% RSLogix 500 project G01098.RSS, saved by version 8.10.00.18 %
PROJECT "G01098"    % processor: SLC 500, 1747-L542 %

PROGRAM FILES
  LAD 2   30 rungs
  LAD 4   21 rungs
  LAD 5   16 rungs
  LAD 20   18 rungs
  LAD 25   24 rungs
  LAD 28   18 rungs
  LAD 29   60 rungs
  LAD 30   13 rungs
  LAD 31   63 rungs
  LAD 32   32 rungs
  LAD 33   10 rungs
  LAD 34   57 rungs
  LAD 35   6 rungs
  LAD 36   5 rungs
  LAD 37   16 rungs
  LAD 38   18 rungs
  LAD 39   59 rungs
  LAD 40   66 rungs
  LAD 50   21 rungs
  LAD 75   16 rungs
  LAD 77   16 rungs
  LAD 80   16 rungs
  LAD 85   37 rungs
  LAD 100   11 rungs
  LAD 101   13 rungs
  LAD 102   14 rungs
  LAD 103   3 rungs
  LAD 110   5 rungs
  LAD 200   24 rungs

DATA FILES
  O0 OUTPUT  23 elements
  I1 INPUT  19 elements
  S2 STATUS  164 elements
  B3 BINARY  105 elements
  T4 TIMER  91 elements
  C5 COUNTER  10 elements
  R6 CONTROL  1 elements
  N7 INTEGER  110 elements
  F8 FLOAT  10 elements
  N10   100 elements
  N11   100 elements
  F15   20 elements
  N20   30 elements
  N30   70 elements
  B33   5 elements
  B34   5 elements
  B50   100 elements
  B51   50 elements
  N52   70 elements
  N53   100 elements
  F54   10 elements
  F55   10 elements
  B56   1 elements
  N58   20 elements
  N59   134 elements
  N60   15 elements
  N61   30 elements
  B94   1 elements
  B95   1 elements
  B96   1 elements
  B97   1 elements
  B98   1 elements
  B99   1 elements
  F197   22 elements
  F198   22 elements
  F199   22 elements
  F200   22 elements
  F201   22 elements
  F202   22 elements
  F203   22 elements
  F204   22 elements
  F205   22 elements
  F206   22 elements
  F207   22 elements
  F208   22 elements
  F209   22 elements
  F210   22 elements
  F211   22 elements
  F212   22 elements
  F213   22 elements
  F214   22 elements
  F215   22 elements
  F216   22 elements
  F217   22 elements
  F218   22 elements
  F219   22 elements
  F220   22 elements
  F221   22 elements
  F222   22 elements
  F223   22 elements
  F224   22 elements
  F225   22 elements
  F226   22 elements
  F227   22 elements
  F228   22 elements
  F229   22 elements
  F230   22 elements
  F231   22 elements
  F232   22 elements
  F233   22 elements
  F234   22 elements
  F235   22 elements
  F236   22 elements
  F237   22 elements
  F238   22 elements
  F239   22 elements
  F240   22 elements
  F241   22 elements
  F242   22 elements
  F243   22 elements
  F244   22 elements
  F245   22 elements
  F246   22 elements
  F247   22 elements
  F248   22 elements
  F249   22 elements
  F250   22 elements

LADDER 2
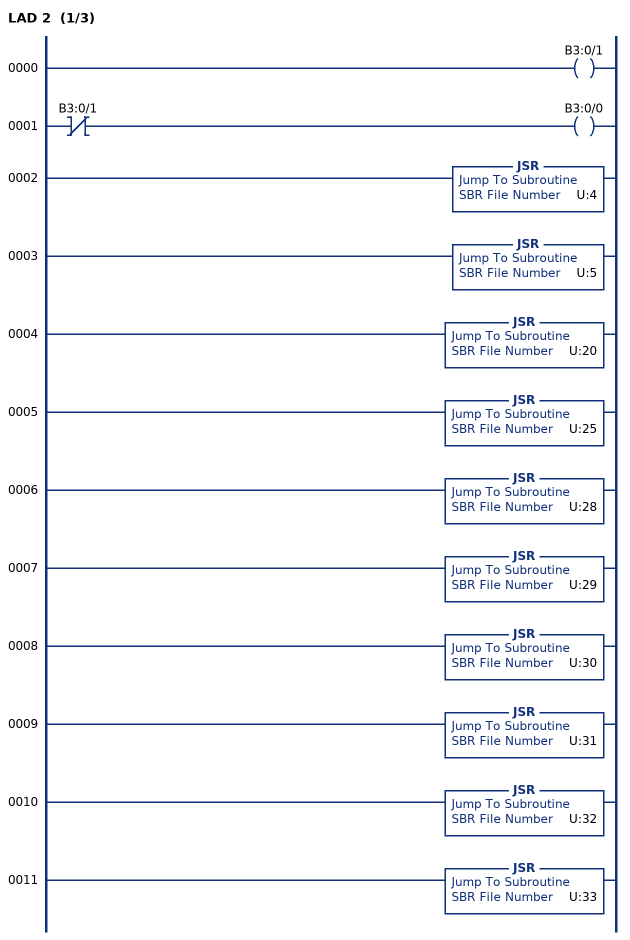
% Rung: 0 %
SOR OTE B3:0/1 EOR
% Rung: 1 %
SOR XIO B3:0/1 OTE B3:0/0 EOR
% Rung: 2 %
SOR JSR U:4 EOR
% Rung: 3 %
SOR JSR U:5 EOR
% Rung: 4 %
SOR JSR U:20 EOR
% Rung: 5 %
SOR JSR U:25 EOR
% Rung: 6 %
SOR JSR U:28 EOR
% Rung: 7 %
SOR JSR U:29 EOR
% Rung: 8 %
SOR JSR U:30 EOR
% Rung: 9 %
SOR JSR U:31 EOR
% Rung: 10 %
SOR JSR U:32 EOR
% Rung: 11 %
SOR JSR U:33 EOR

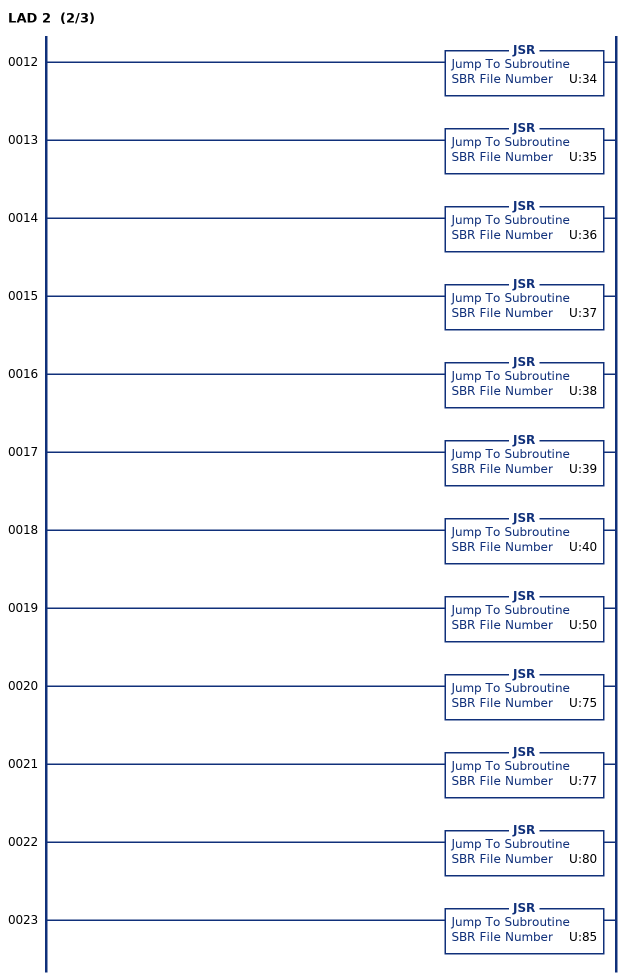
% Rung: 12 %
SOR JSR U:34 EOR
% Rung: 13 %
SOR JSR U:35 EOR
% Rung: 14 %
SOR JSR U:36 EOR
% Rung: 15 %
SOR JSR U:37 EOR
% Rung: 16 %
SOR JSR U:38 EOR
% Rung: 17 %
SOR JSR U:39 EOR
% Rung: 18 %
SOR JSR U:40 EOR
% Rung: 19 %
SOR JSR U:50 EOR
% Rung: 20 %
SOR JSR U:75 EOR
% Rung: 21 %
SOR JSR U:77 EOR
% Rung: 22 %
SOR JSR U:80 EOR
% Rung: 23 %
SOR JSR U:85 EOR

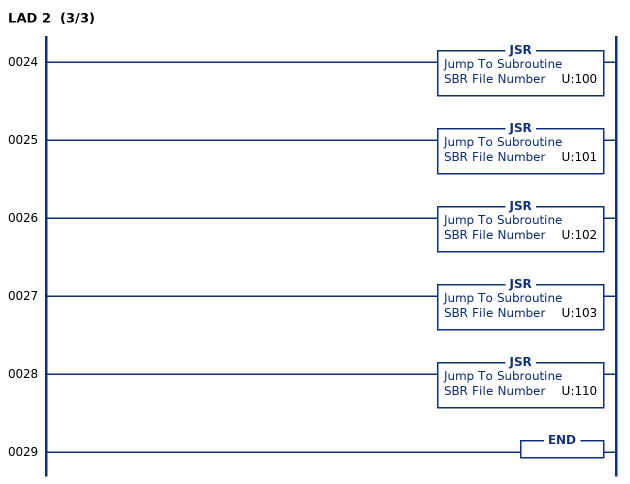
% Rung: 24 %
SOR JSR U:100 EOR
% Rung: 25 %
SOR JSR U:101 EOR
% Rung: 26 %
SOR JSR U:102 EOR
% Rung: 27 %
SOR JSR U:103 EOR
% Rung: 28 %
SOR JSR U:110 EOR
% Rung: 29 %
SOR END EOR

LADDER 4
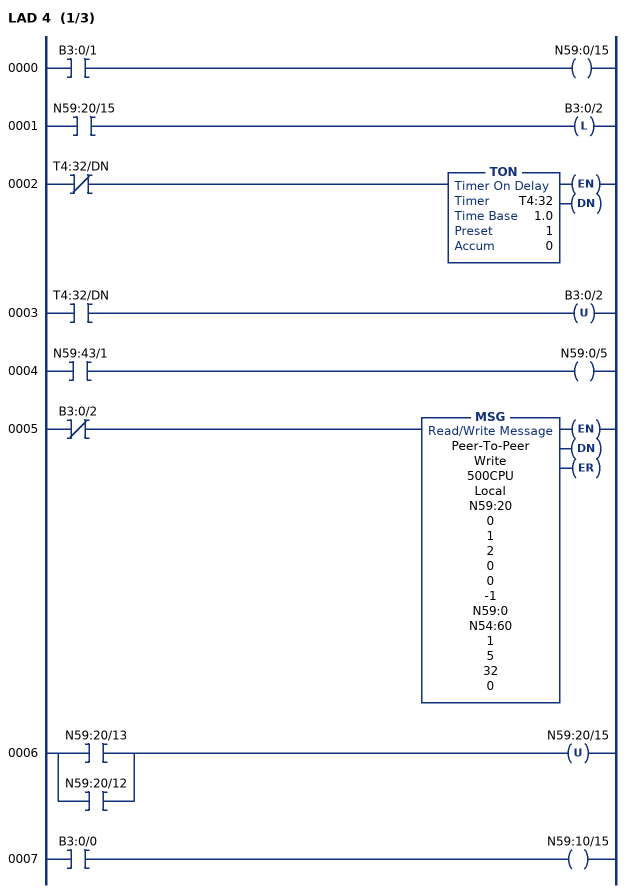
% Rung: 0 %
SOR XIC B3:0/1 OTE N59:0/15 EOR
% Rung: 1 %
SOR XIC N59:20/15 OTL B3:0/2 EOR
% Rung: 2 %
SOR XIO T4:32/DN TON T4:32 1.0 1 0 EOR
% Rung: 3 %
SOR XIC T4:32/DN OTU B3:0/2 EOR
% Rung: 4 %
SOR XIC N59:43/1 OTE N59:0/5 EOR
% Rung: 5 %
SOR XIO B3:0/2 MSG Peer-To-Peer Write 500CPU Local N59:20 0 1 2 0 0 -1 N59:0 N54:60 1 5 32 0 EOR
%   MSG set-up: 500CPU Write | 5 | 1 | N54:60 | N59:0 | 0 | 2 | 2 | CLIENT | 0 | 0 %
% Rung: 6 %
SOR BST XIC N59:20/13 NXB XIC N59:20/12 BND OTU N59:20/15 EOR
% Rung: 7 %
SOR XIC B3:0/0 OTE N59:10/15 EOR

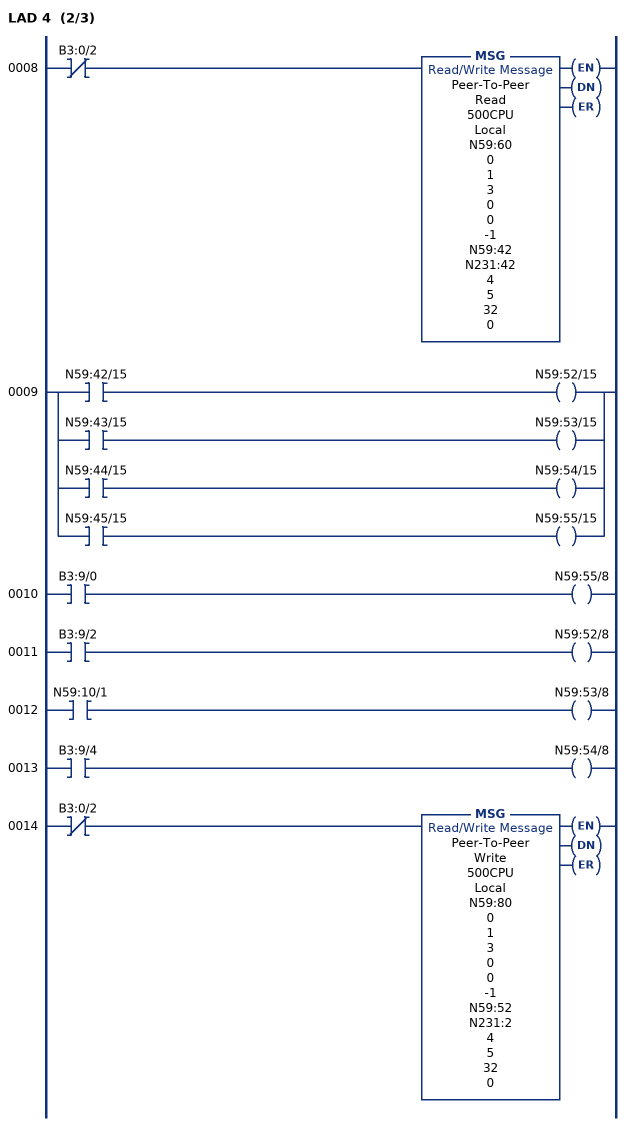
% Rung: 8 %
SOR XIO B3:0/2 MSG Peer-To-Peer Read 500CPU Local N59:60 0 1 3 0 0 -1 N59:42 N231:42 4 5 32 0 EOR
%   MSG set-up: 500CPU Read | 5 | 4 | N231:42 | N59:42 | 0 | 3 | 3 | CLIENT | 0 | 0 %
% Rung: 9 %
SOR BST XIC N59:42/15 OTE N59:52/15 NXB XIC N59:43/15 OTE N59:53/15 NXB XIC N59:44/15 OTE N59:54/15 NXB XIC N59:45/15 OTE N59:55/15 BND EOR
% Rung: 10 %
SOR XIC B3:9/0 OTE N59:55/8 EOR
% Rung: 11 %
SOR XIC B3:9/2 OTE N59:52/8 EOR
% Rung: 12 %
SOR XIC N59:10/1 OTE N59:53/8 EOR
% Rung: 13 %
SOR XIC B3:9/4 OTE N59:54/8 EOR
% Rung: 14 %
SOR XIO B3:0/2 MSG Peer-To-Peer Write 500CPU Local N59:80 0 1 3 0 0 -1 N59:52 N231:2 4 5 32 0 EOR
%   MSG set-up: 500CPU Write | 5 | 4 | N231:2 | N59:52 | 0 | 3 | 3 | CLIENT | 0 | 0 %

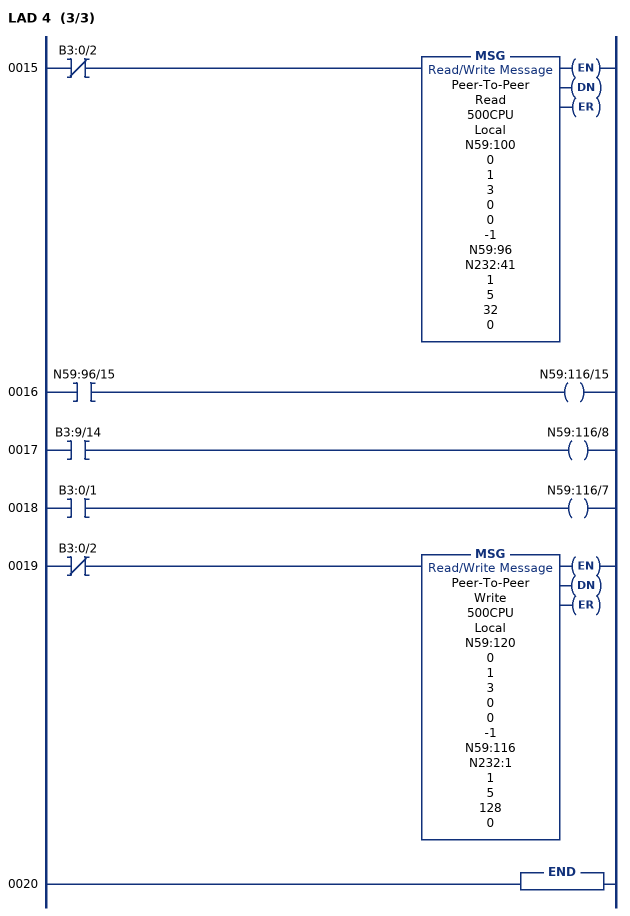
% Rung: 15 %
SOR XIO B3:0/2 MSG Peer-To-Peer Read 500CPU Local N59:100 0 1 3 0 0 -1 N59:96 N232:41 1 5 32 0 EOR
%   MSG set-up: 500CPU Read | 5 | 1 | N232:41 | N59:96 | 0 | 3 | 3 | CLIENT | 0 | 0 %
% Rung: 16 %
SOR XIC N59:96/15 OTE N59:116/15 EOR
% Rung: 17 %
SOR XIC B3:9/14 OTE N59:116/8 EOR
% Rung: 18 %
SOR XIC B3:0/1 OTE N59:116/7 EOR
% Rung: 19 %
SOR XIO B3:0/2 MSG Peer-To-Peer Write 500CPU Local N59:120 0 1 3 0 0 -1 N59:116 N232:1 1 5 128 0 EOR
%   MSG set-up: 500CPU Write | 5 | 1 | N232:1 | N59:116 | 0 | 3 | 3 | CLIENT | 0 | 0 %
% Rung: 20 %
SOR END EOR

LADDER 5
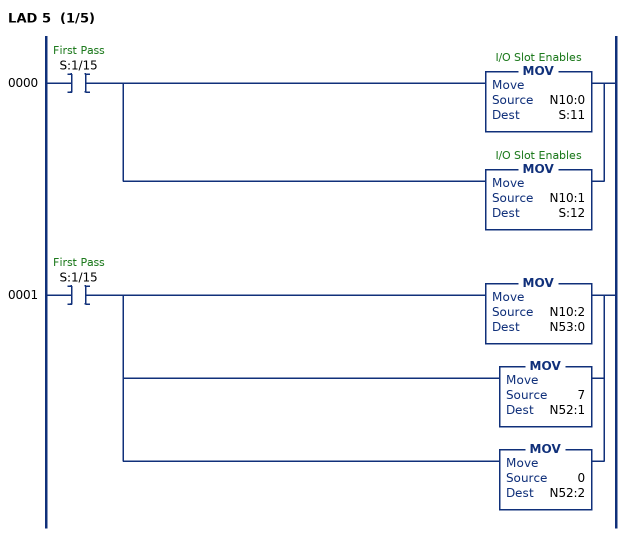
% Rung: 0 %
SOR XIC S:1/15 BST MOV N10:0 S:11 NXB MOV N10:1 S:12 BND EOR
%   S:1/15  "First Pass" %
%   S:11  "I/O Slot Enables" %
%   S:12  "I/O Slot Enables" %
% Rung: 1 %
SOR XIC S:1/15 BST MOV N10:2 N53:0 NXB MOV 7 N52:1 NXB MOV 0 N52:2 BND EOR
%   S:1/15  "First Pass" %

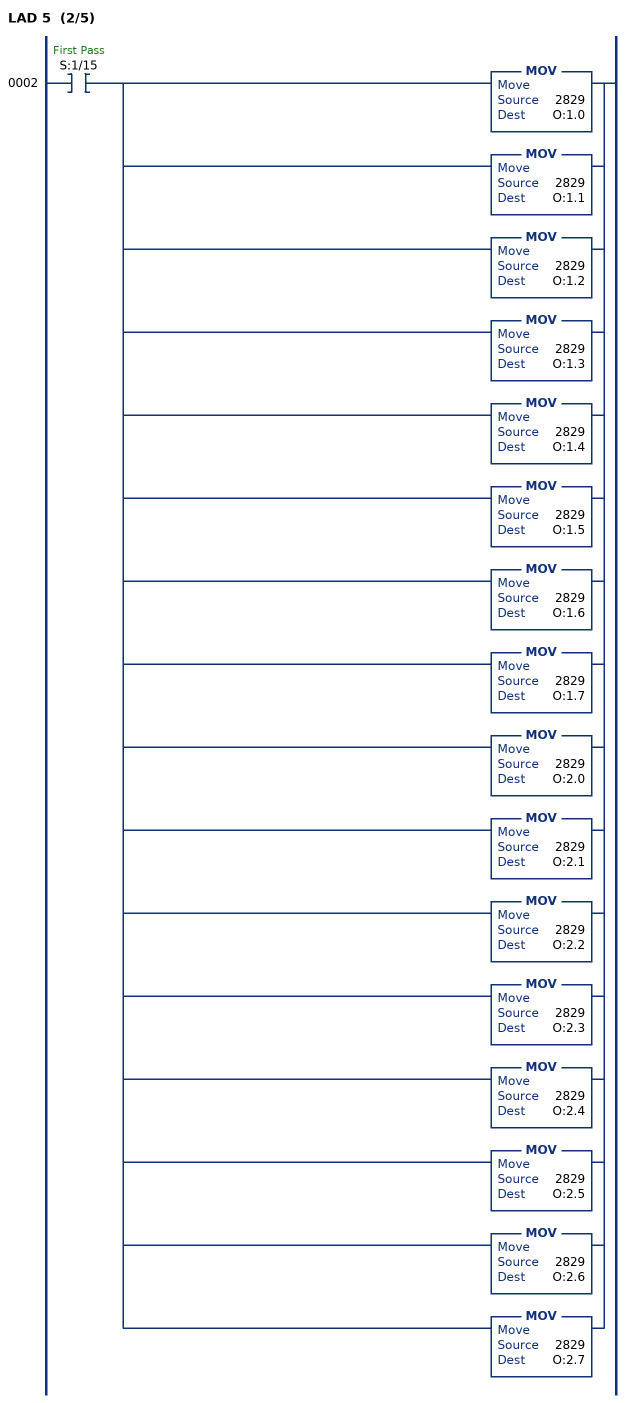
% Rung: 2 %
SOR XIC S:1/15 BST MOV 2829 O:1.0 NXB MOV 2829 O:1.1 NXB MOV 2829 O:1.2 NXB MOV 2829 O:1.3 NXB MOV 2829 O:1.4 NXB MOV 2829 O:1.5 NXB MOV 2829 O:1.6 NXB MOV 2829 O:1.7 NXB MOV 2829 O:2.0 NXB MOV 2829 O:2.1 NXB MOV 2829 O:2.2 NXB MOV 2829 O:2.3 NXB MOV 2829 O:2.4 NXB MOV 2829 O:2.5 NXB MOV 2829 O:2.6 NXB MOV 2829 O:2.7 BND EOR
%   S:1/15  "First Pass" %

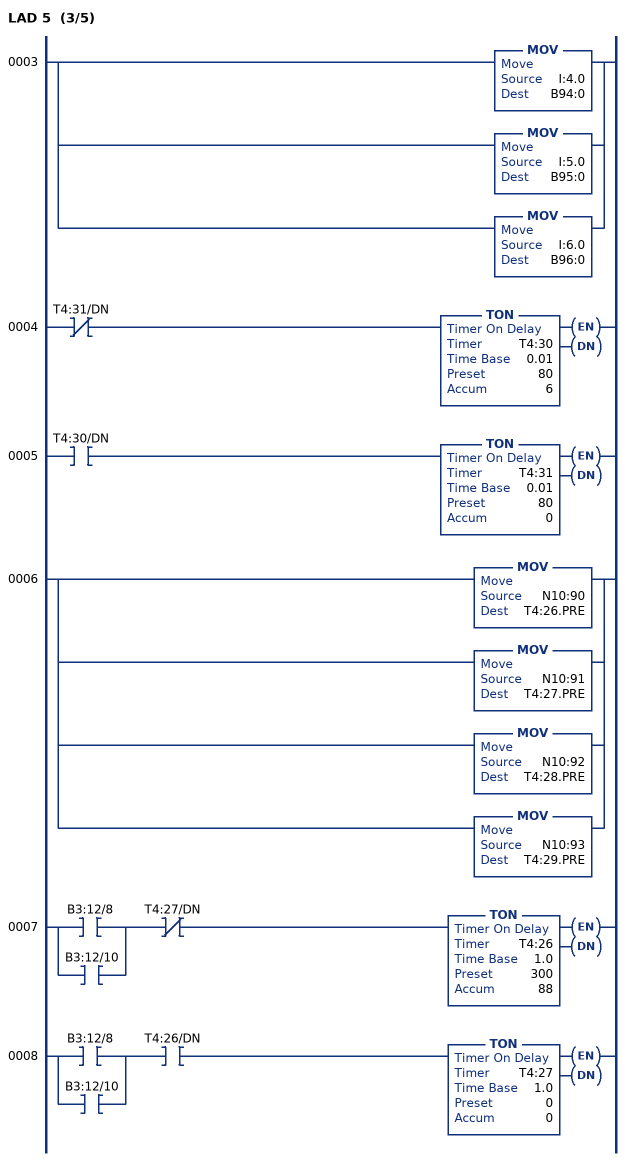
% Rung: 3 %
SOR BST MOV I:4.0 B94:0 NXB MOV I:5.0 B95:0 NXB MOV I:6.0 B96:0 BND EOR
% Rung: 4 %
SOR XIO T4:31/DN TON T4:30 0.01 80 6 EOR
% Rung: 5 %
SOR XIC T4:30/DN TON T4:31 0.01 80 0 EOR
% Rung: 6 %
SOR BST MOV N10:90 T4:26.PRE NXB MOV N10:91 T4:27.PRE NXB MOV N10:92 T4:28.PRE NXB MOV N10:93 T4:29.PRE BND EOR
% Rung: 7 %
SOR BST XIC B3:12/8 NXB XIC B3:12/10 BND XIO T4:27/DN TON T4:26 1.0 300 88 EOR
% Rung: 8 %
SOR BST XIC B3:12/8 NXB XIC B3:12/10 BND XIC T4:26/DN TON T4:27 1.0 0 0 EOR

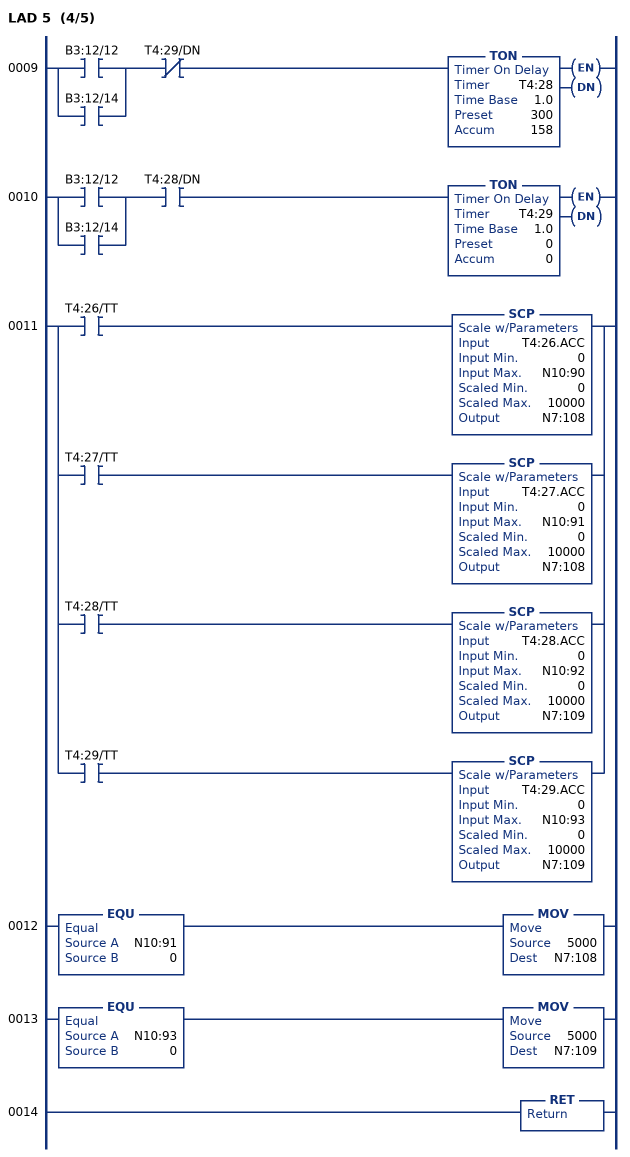
% Rung: 9 %
SOR BST XIC B3:12/12 NXB XIC B3:12/14 BND XIO T4:29/DN TON T4:28 1.0 300 158 EOR
% Rung: 10 %
SOR BST XIC B3:12/12 NXB XIC B3:12/14 BND XIC T4:28/DN TON T4:29 1.0 0 0 EOR
% Rung: 11 %
SOR BST XIC T4:26/TT SCP T4:26.ACC 0 N10:90 0 10000 N7:108 NXB XIC T4:27/TT SCP T4:27.ACC 0 N10:91 0 10000 N7:108 NXB XIC T4:28/TT SCP T4:28.ACC 0 N10:92 0 10000 N7:109 NXB XIC T4:29/TT SCP T4:29.ACC 0 N10:93 0 10000 N7:109 BND EOR
% Rung: 12 %
SOR EQU N10:91 0 MOV 5000 N7:108 EOR
% Rung: 13 %
SOR EQU N10:93 0 MOV 5000 N7:109 EOR
% Rung: 14 %
SOR RET EOR

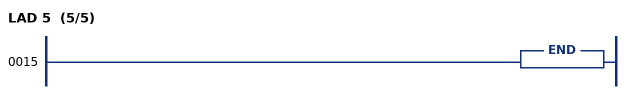
% Rung: 15 %
SOR END EOR

LADDER 20
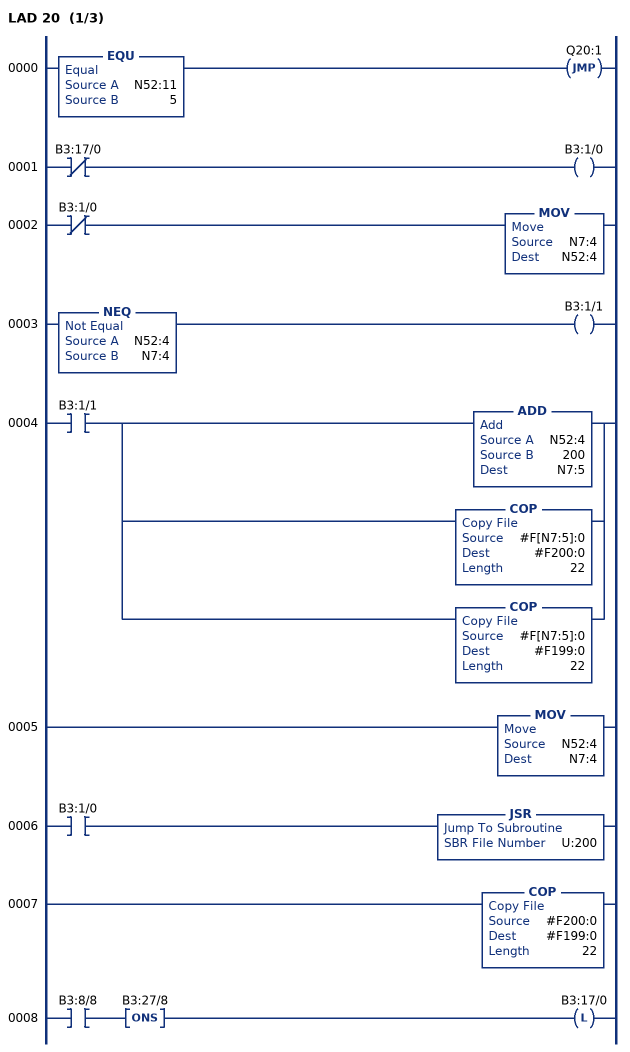
% Rung: 0 %
SOR EQU N52:11 5 JMP Q20:1 EOR
% Rung: 1 %
SOR XIO B3:17/0 OTE B3:1/0 EOR
% Rung: 2 %
SOR XIO B3:1/0 MOV N7:4 N52:4 EOR
% Rung: 3 %
SOR NEQ N52:4 N7:4 OTE B3:1/1 EOR
% Rung: 4 %
SOR XIC B3:1/1 BST ADD N52:4 200 N7:5 NXB COP #F[N7:5]:0 #F200:0 22 NXB COP #F[N7:5]:0 #F199:0 22 BND EOR
% Rung: 5 %
SOR MOV N52:4 N7:4 EOR
% Rung: 6 %
SOR XIC B3:1/0 JSR U:200 EOR
% Rung: 7 %
SOR COP #F200:0 #F199:0 22 EOR
% Rung: 8 %
SOR XIC B3:8/8 OSR B3:27/8 OTL B3:17/0 EOR

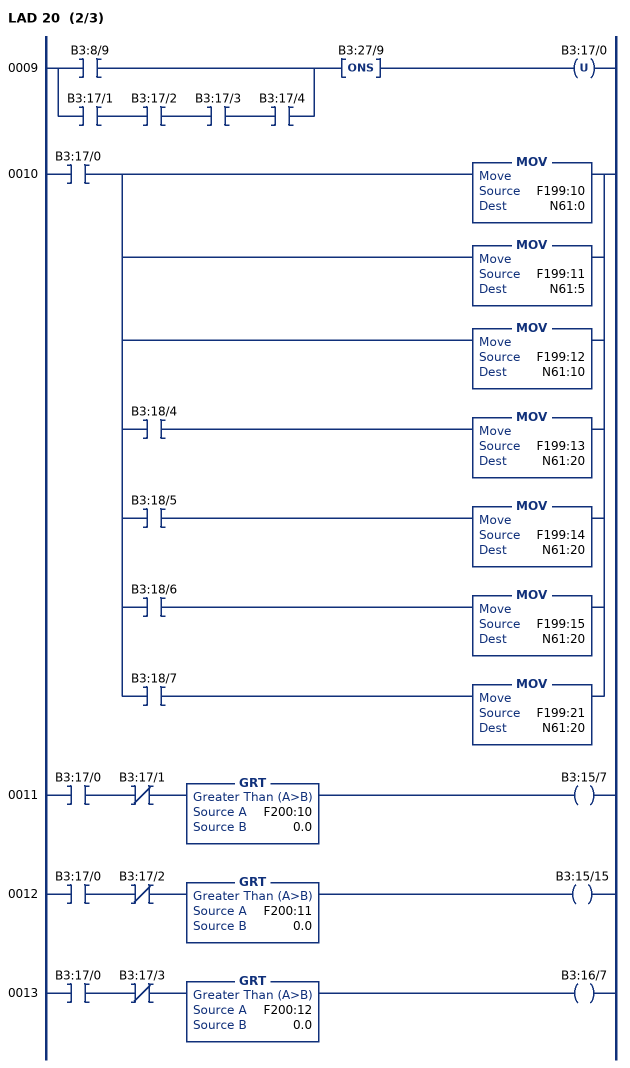
% Rung: 9 %
SOR BST XIC B3:8/9 NXB XIC B3:17/1 XIC B3:17/2 XIC B3:17/3 XIC B3:17/4 BND OSR B3:27/9 OTU B3:17/0 EOR
% Rung: 10 %
SOR XIC B3:17/0 BST MOV F199:10 N61:0 NXB MOV F199:11 N61:5 NXB MOV F199:12 N61:10 NXB XIC B3:18/4 MOV F199:13 N61:20 NXB XIC B3:18/5 MOV F199:14 N61:20 NXB XIC B3:18/6 MOV F199:15 N61:20 NXB XIC B3:18/7 MOV F199:21 N61:20 BND EOR
% Rung: 11 %
SOR XIC B3:17/0 XIO B3:17/1 GRT F200:10 0.0 OTE B3:15/7 EOR
% Rung: 12 %
SOR XIC B3:17/0 XIO B3:17/2 GRT F200:11 0.0 OTE B3:15/15 EOR
% Rung: 13 %
SOR XIC B3:17/0 XIO B3:17/3 GRT F200:12 0.0 OTE B3:16/7 EOR

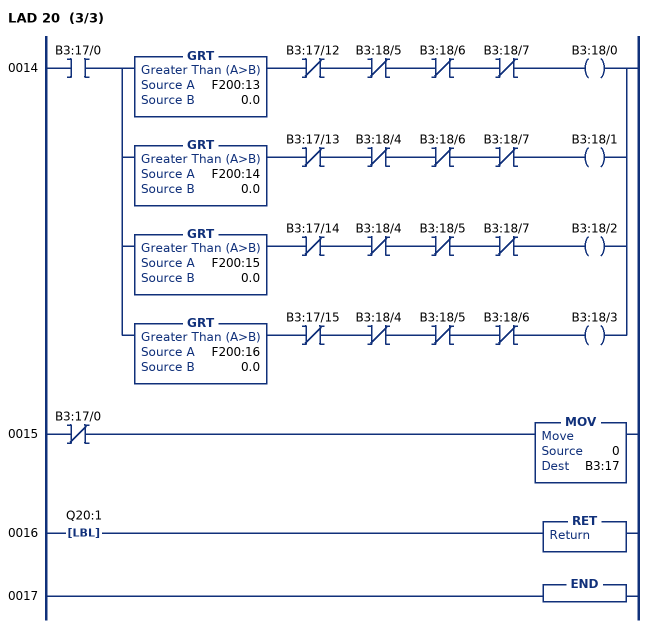
% Rung: 14 %
SOR XIC B3:17/0 BST GRT F200:13 0.0 XIO B3:17/12 XIO B3:18/5 XIO B3:18/6 XIO B3:18/7 OTE B3:18/0 NXB GRT F200:14 0.0 XIO B3:17/13 XIO B3:18/4 XIO B3:18/6 XIO B3:18/7 OTE B3:18/1 NXB GRT F200:15 0.0 XIO B3:17/14 XIO B3:18/4 XIO B3:18/5 XIO B3:18/7 OTE B3:18/2 NXB GRT F200:16 0.0 XIO B3:17/15 XIO B3:18/4 XIO B3:18/5 XIO B3:18/6 OTE B3:18/3 BND EOR
% Rung: 15 %
SOR XIO B3:17/0 MOV 0 B3:17 EOR
% Rung: 16 %
SOR LBL Q20:1 RET EOR
% Rung: 17 %
SOR END EOR

LADDER 25
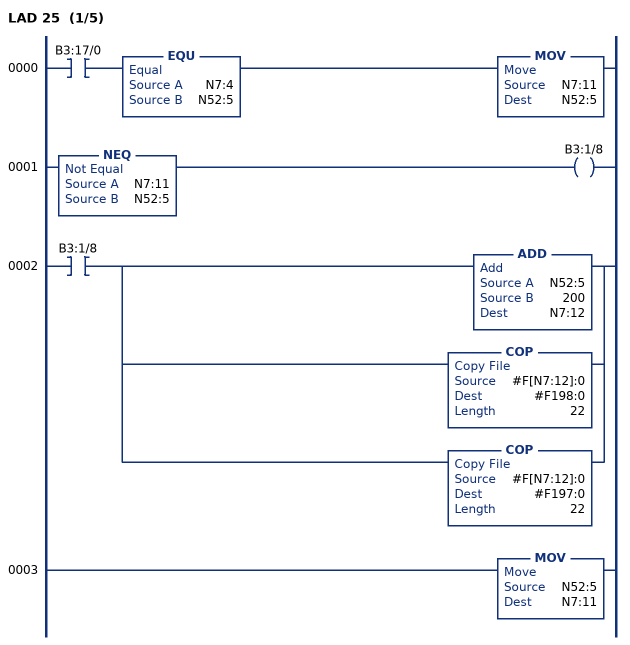
% Rung: 0 %
SOR XIC B3:17/0 EQU N7:4 N52:5 MOV N7:11 N52:5 EOR
% Rung: 1 %
SOR NEQ N7:11 N52:5 OTE B3:1/8 EOR
% Rung: 2 %
SOR XIC B3:1/8 BST ADD N52:5 200 N7:12 NXB COP #F[N7:12]:0 #F198:0 22 NXB COP #F[N7:12]:0 #F197:0 22 BND EOR
% Rung: 3 %
SOR MOV N52:5 N7:11 EOR

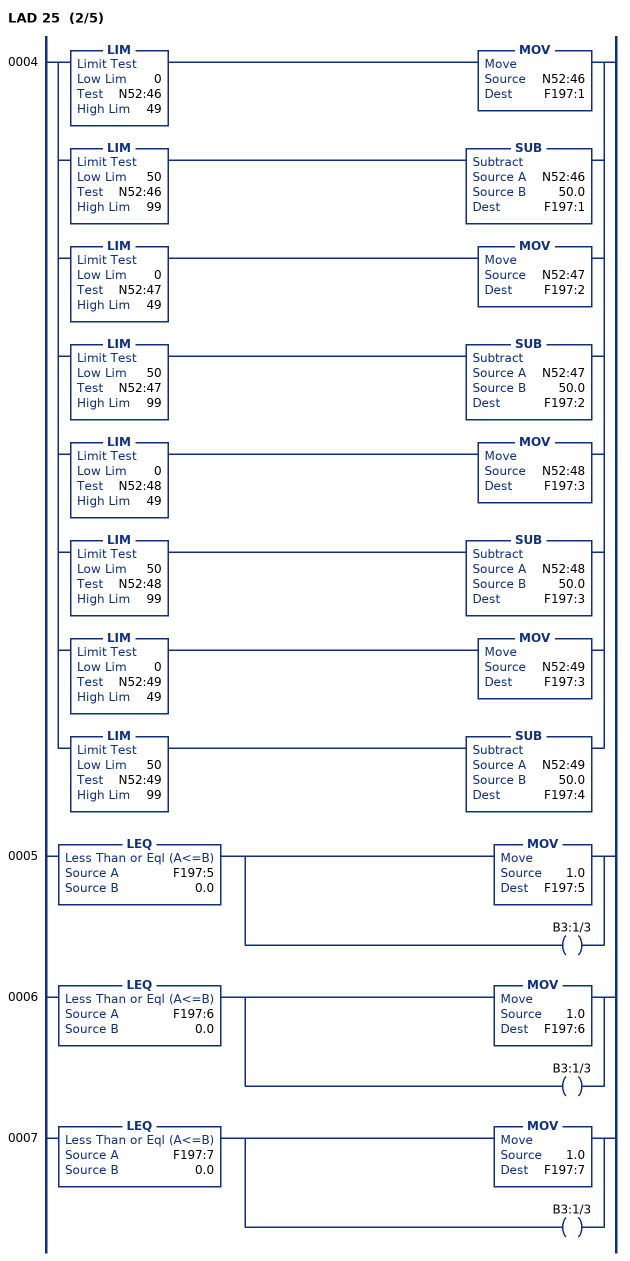
% Rung: 4 %
SOR BST LIM 0 N52:46 49 MOV N52:46 F197:1 NXB LIM 50 N52:46 99 SUB N52:46 50.0 F197:1 NXB LIM 0 N52:47 49 MOV N52:47 F197:2 NXB LIM 50 N52:47 99 SUB N52:47 50.0 F197:2 NXB LIM 0 N52:48 49 MOV N52:48 F197:3 NXB LIM 50 N52:48 99 SUB N52:48 50.0 F197:3 NXB LIM 0 N52:49 49 MOV N52:49 F197:3 NXB LIM 50 N52:49 99 SUB N52:49 50.0 F197:4 BND EOR
% Rung: 5 %
SOR LEQ F197:5 0.0 BST MOV 1.0 F197:5 NXB OTE B3:1/3 BND EOR
% Rung: 6 %
SOR LEQ F197:6 0.0 BST MOV 1.0 F197:6 NXB OTE B3:1/3 BND EOR
% Rung: 7 %
SOR LEQ F197:7 0.0 BST MOV 1.0 F197:7 NXB OTE B3:1/3 BND EOR

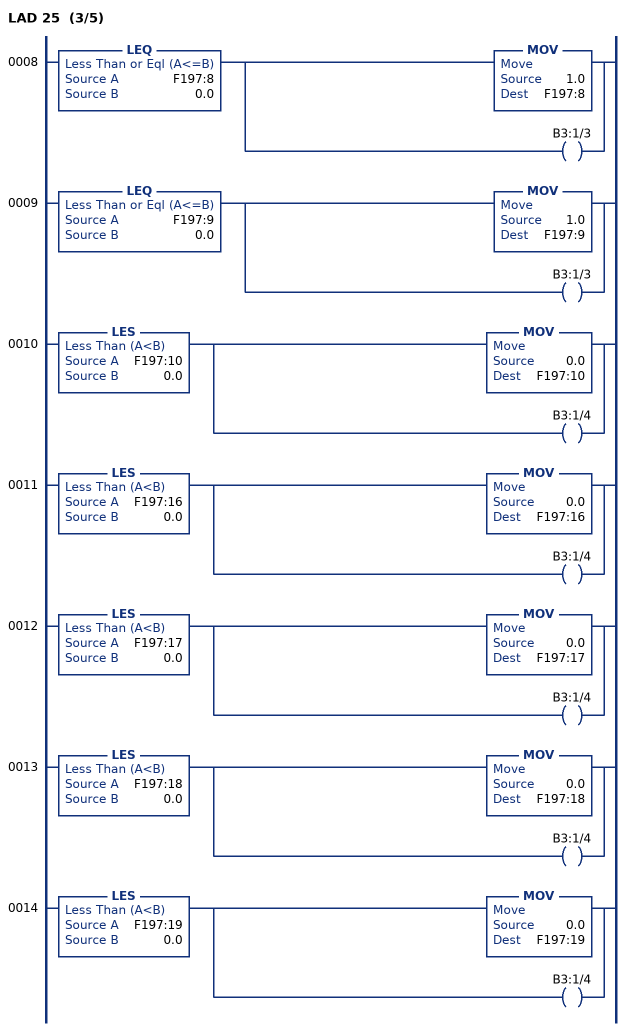
% Rung: 8 %
SOR LEQ F197:8 0.0 BST MOV 1.0 F197:8 NXB OTE B3:1/3 BND EOR
% Rung: 9 %
SOR LEQ F197:9 0.0 BST MOV 1.0 F197:9 NXB OTE B3:1/3 BND EOR
% Rung: 10 %
SOR LES F197:10 0.0 BST MOV 0.0 F197:10 NXB OTE B3:1/4 BND EOR
% Rung: 11 %
SOR LES F197:16 0.0 BST MOV 0.0 F197:16 NXB OTE B3:1/4 BND EOR
% Rung: 12 %
SOR LES F197:17 0.0 BST MOV 0.0 F197:17 NXB OTE B3:1/4 BND EOR
% Rung: 13 %
SOR LES F197:18 0.0 BST MOV 0.0 F197:18 NXB OTE B3:1/4 BND EOR
% Rung: 14 %
SOR LES F197:19 0.0 BST MOV 0.0 F197:19 NXB OTE B3:1/4 BND EOR

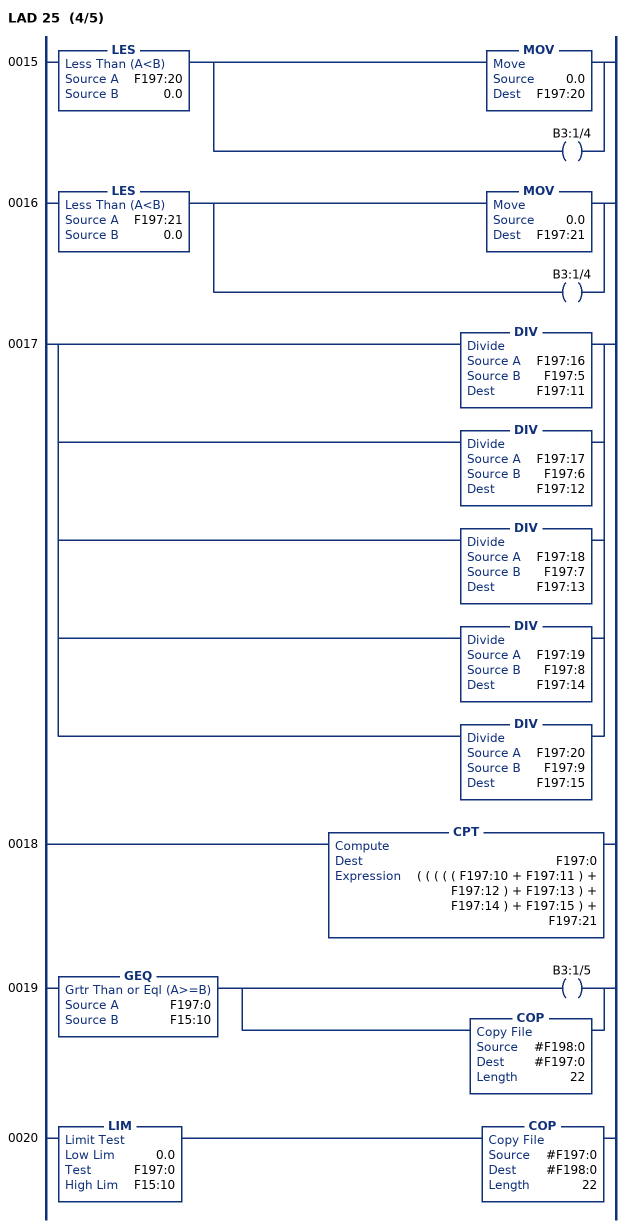
% Rung: 15 %
SOR LES F197:20 0.0 BST MOV 0.0 F197:20 NXB OTE B3:1/4 BND EOR
% Rung: 16 %
SOR LES F197:21 0.0 BST MOV 0.0 F197:21 NXB OTE B3:1/4 BND EOR
% Rung: 17 %
SOR BST DIV F197:16 F197:5 F197:11 NXB DIV F197:17 F197:6 F197:12 NXB DIV F197:18 F197:7 F197:13 NXB DIV F197:19 F197:8 F197:14 NXB DIV F197:20 F197:9 F197:15 BND EOR
% Rung: 18 %
SOR CPT F197:0 " ( ( ( ( ( F197:10 + F197:11 ) + F197:12 ) + F197:13 ) + F197:14 ) + F197:15 ) + F197:21 " EOR
% Rung: 19 %
SOR GEQ F197:0 F15:10 BST OTE B3:1/5 NXB COP #F198:0 #F197:0 22 BND EOR
% Rung: 20 %
SOR LIM 0.0 F197:0 F15:10 COP #F197:0 #F198:0 22 EOR

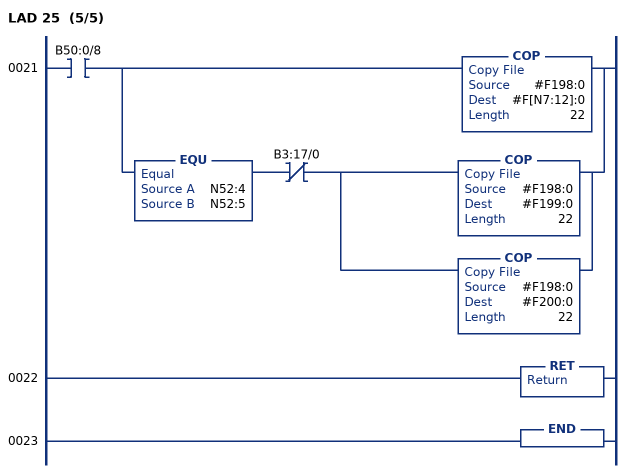
% Rung: 21 %
SOR XIC B50:0/8 BST COP #F198:0 #F[N7:12]:0 22 NXB EQU N52:4 N52:5 XIO B3:17/0 BST COP #F198:0 #F199:0 22 NXB COP #F198:0 #F200:0 22 BND BND EOR
% Rung: 22 %
SOR RET EOR
% Rung: 23 %
SOR END EOR

LADDER 28
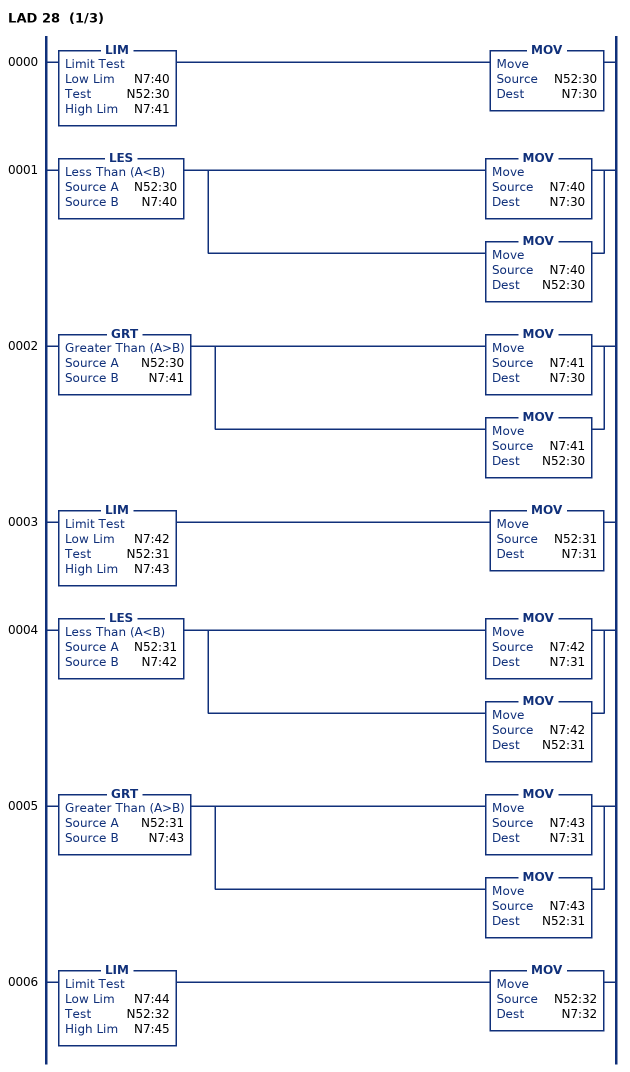
% Rung: 0 %
SOR LIM N7:40 N52:30 N7:41 MOV N52:30 N7:30 EOR
% Rung: 1 %
SOR LES N52:30 N7:40 BST MOV N7:40 N7:30 NXB MOV N7:40 N52:30 BND EOR
% Rung: 2 %
SOR GRT N52:30 N7:41 BST MOV N7:41 N7:30 NXB MOV N7:41 N52:30 BND EOR
% Rung: 3 %
SOR LIM N7:42 N52:31 N7:43 MOV N52:31 N7:31 EOR
% Rung: 4 %
SOR LES N52:31 N7:42 BST MOV N7:42 N7:31 NXB MOV N7:42 N52:31 BND EOR
% Rung: 5 %
SOR GRT N52:31 N7:43 BST MOV N7:43 N7:31 NXB MOV N7:43 N52:31 BND EOR
% Rung: 6 %
SOR LIM N7:44 N52:32 N7:45 MOV N52:32 N7:32 EOR

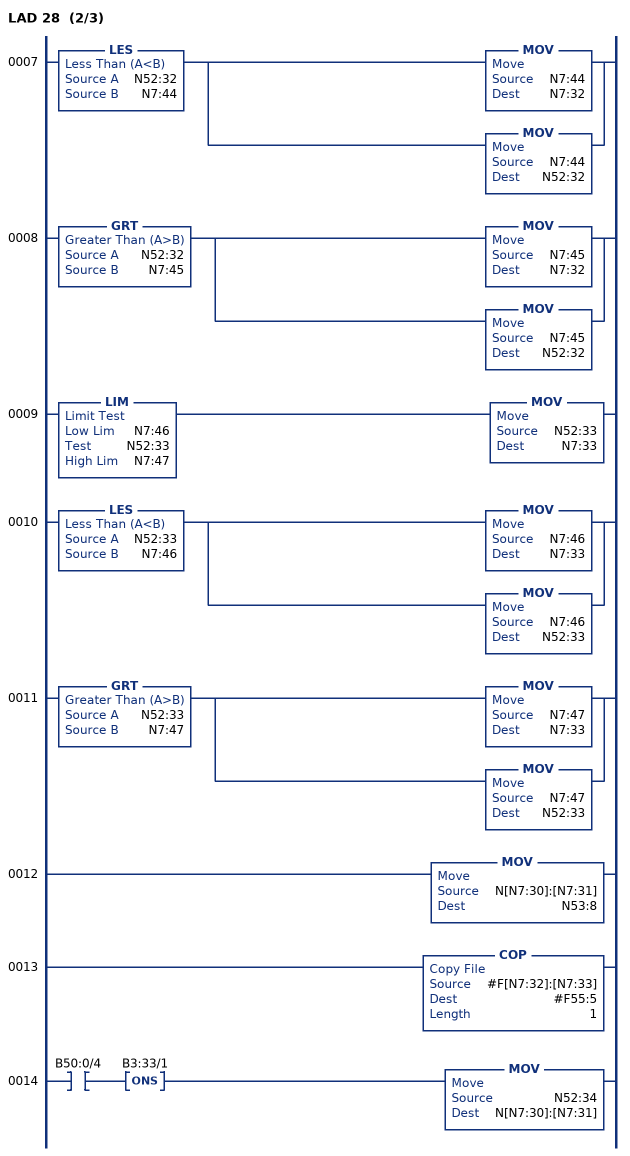
% Rung: 7 %
SOR LES N52:32 N7:44 BST MOV N7:44 N7:32 NXB MOV N7:44 N52:32 BND EOR
% Rung: 8 %
SOR GRT N52:32 N7:45 BST MOV N7:45 N7:32 NXB MOV N7:45 N52:32 BND EOR
% Rung: 9 %
SOR LIM N7:46 N52:33 N7:47 MOV N52:33 N7:33 EOR
% Rung: 10 %
SOR LES N52:33 N7:46 BST MOV N7:46 N7:33 NXB MOV N7:46 N52:33 BND EOR
% Rung: 11 %
SOR GRT N52:33 N7:47 BST MOV N7:47 N7:33 NXB MOV N7:47 N52:33 BND EOR
% Rung: 12 %
SOR MOV N[N7:30]:[N7:31] N53:8 EOR
% Rung: 13 %
SOR COP #F[N7:32]:[N7:33] #F55:5 1 EOR
% Rung: 14 %
SOR XIC B50:0/4 OSR B3:33/1 MOV N52:34 N[N7:30]:[N7:31] EOR

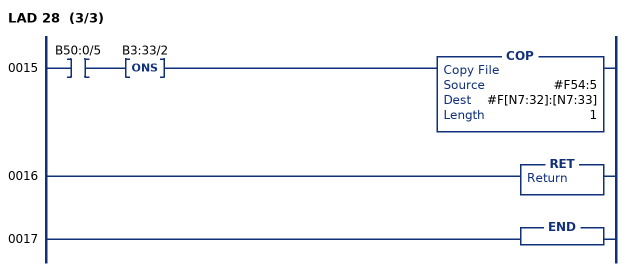
% Rung: 15 %
SOR XIC B50:0/5 OSR B3:33/2 COP #F54:5 #F[N7:32]:[N7:33] 1 EOR
% Rung: 16 %
SOR RET EOR
% Rung: 17 %
SOR END EOR

LADDER 29
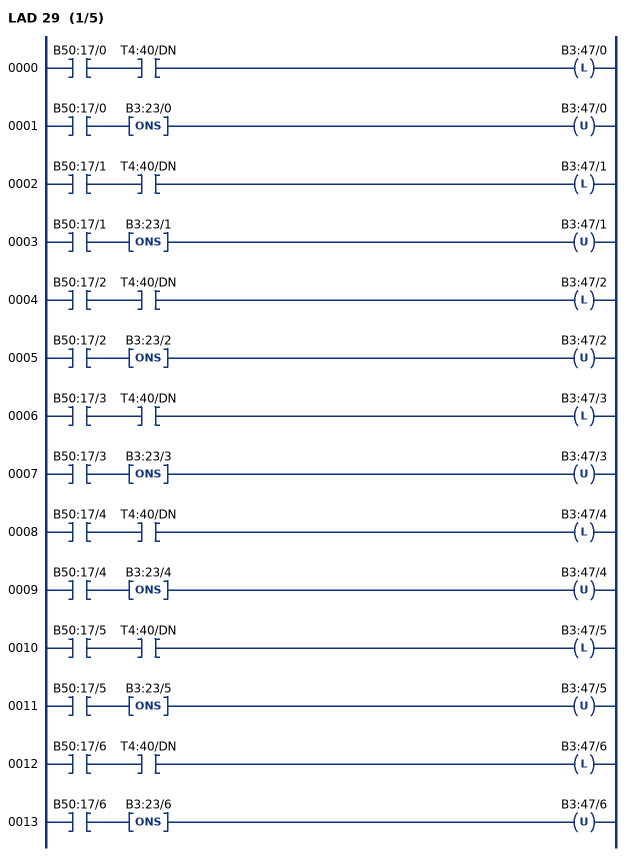
% Rung: 0 %
SOR XIC B50:17/0 XIC T4:40/DN OTL B3:47/0 EOR
% Rung: 1 %
SOR XIC B50:17/0 OSR B3:23/0 OTU B3:47/0 EOR
% Rung: 2 %
SOR XIC B50:17/1 XIC T4:40/DN OTL B3:47/1 EOR
% Rung: 3 %
SOR XIC B50:17/1 OSR B3:23/1 OTU B3:47/1 EOR
% Rung: 4 %
SOR XIC B50:17/2 XIC T4:40/DN OTL B3:47/2 EOR
% Rung: 5 %
SOR XIC B50:17/2 OSR B3:23/2 OTU B3:47/2 EOR
% Rung: 6 %
SOR XIC B50:17/3 XIC T4:40/DN OTL B3:47/3 EOR
% Rung: 7 %
SOR XIC B50:17/3 OSR B3:23/3 OTU B3:47/3 EOR
% Rung: 8 %
SOR XIC B50:17/4 XIC T4:40/DN OTL B3:47/4 EOR
% Rung: 9 %
SOR XIC B50:17/4 OSR B3:23/4 OTU B3:47/4 EOR
% Rung: 10 %
SOR XIC B50:17/5 XIC T4:40/DN OTL B3:47/5 EOR
% Rung: 11 %
SOR XIC B50:17/5 OSR B3:23/5 OTU B3:47/5 EOR
% Rung: 12 %
SOR XIC B50:17/6 XIC T4:40/DN OTL B3:47/6 EOR
% Rung: 13 %
SOR XIC B50:17/6 OSR B3:23/6 OTU B3:47/6 EOR

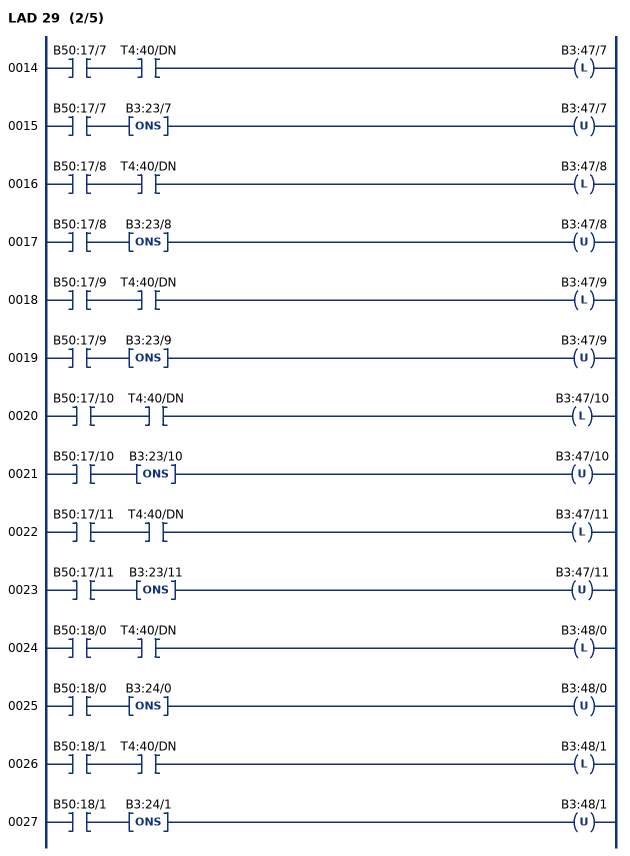
% Rung: 14 %
SOR XIC B50:17/7 XIC T4:40/DN OTL B3:47/7 EOR
% Rung: 15 %
SOR XIC B50:17/7 OSR B3:23/7 OTU B3:47/7 EOR
% Rung: 16 %
SOR XIC B50:17/8 XIC T4:40/DN OTL B3:47/8 EOR
% Rung: 17 %
SOR XIC B50:17/8 OSR B3:23/8 OTU B3:47/8 EOR
% Rung: 18 %
SOR XIC B50:17/9 XIC T4:40/DN OTL B3:47/9 EOR
% Rung: 19 %
SOR XIC B50:17/9 OSR B3:23/9 OTU B3:47/9 EOR
% Rung: 20 %
SOR XIC B50:17/10 XIC T4:40/DN OTL B3:47/10 EOR
% Rung: 21 %
SOR XIC B50:17/10 OSR B3:23/10 OTU B3:47/10 EOR
% Rung: 22 %
SOR XIC B50:17/11 XIC T4:40/DN OTL B3:47/11 EOR
% Rung: 23 %
SOR XIC B50:17/11 OSR B3:23/11 OTU B3:47/11 EOR
% Rung: 24 %
SOR XIC B50:18/0 XIC T4:40/DN OTL B3:48/0 EOR
% Rung: 25 %
SOR XIC B50:18/0 OSR B3:24/0 OTU B3:48/0 EOR
% Rung: 26 %
SOR XIC B50:18/1 XIC T4:40/DN OTL B3:48/1 EOR
% Rung: 27 %
SOR XIC B50:18/1 OSR B3:24/1 OTU B3:48/1 EOR

